PROGRAM INTERNAL MAIN_TESTS
VAR
	_driveTest : fbDriveTest;
END_VAR

_driveTest();

END_PROGRAM

(* stored: Version 1.1.0.1, ProductVersion 3.1.4024.6
   POU MAIN_TESTS: Id {d1e7ffc5-0e5e-40b6-83db-d6d43156a01c}, SpecialFunc None *)
